// TIA Portal V15 export
// export: Created 2018-12-10T18:36:46.2365966Z, ExportSetting WithDefaults, WithReadOnly, DisplayName Totally Integrated Automation Portal, DisplayVersion V15 Update 2, DisplayName TIA Portal Openness, DisplayVersion V15 Update 2, DisplayName STEP 7 Professional, DisplayVersion V15 Update 2, DisplayName STEP 7 Safety, DisplayVersion V15, DisplayName WinCC Professional, DisplayVersion V15 Update 2, DisplayName SIMATIC Visualization Architect, DisplayVersion V15 Update 1
DATA_BLOCK "FGDB_ROBNAME@FlowDrill"   // DB118
TITLE = Tehchnology flow drill / Technologie übergreifendes Gerät
{ S7_Optimized_Access := 'FALSE' }
AUTHOR : integra
FAMILY : SUB
VERSION : 0.1
// stored: AutoNumber true, CodeModifiedDate 2018-02-20T07:56:40.7852281Z, CompileDate 2018-02-20T10:24:49.1738274Z, CreationDate 2017-02-23T12:13:10.5636609Z, DBAccessibleFromOPCUA true, InstanceOfName iSF_TECH_ROBOT_FLOW_DRILL_SCREWING, InstanceOfNumber 24, InstanceOfType FB, InterfaceModifiedDate 2018-02-19T12:53:42.2863137Z, IsConsistent true, IsKnowHowProtected false, ModifiedDate 2018-02-20T07:56:40.7852281Z, ParameterModified 2018-02-19T12:53:31.0081644Z, StructureModified 2018-02-19T12:53:42.2863137Z, UDAEnableTagReadback false
"iSF_TECH_ROBOT_FLOW_DRILL_SCREWING"
   // VAR_INPUT
   //    fct : Int;
   //    safetyStop : Bool;
   //    functionPoint : String[6];
   //    identType : String[12];
   // END_VAR
   // VAR_OUTPUT
   //    counterParts : Int;
   //    counterNIOpoints : Int;
   //    counterIOpoints : Int;
   //    fault : Bool;
   // END_VAR
   // VAR_IN_OUT
   //    IfcFGExternal : "iUDT_IFC_SYS_EXTERNAL_ALARM";
   //    IfcTECH : "iUDT_IFC_ROBOT_TECH";
   //    IfcAcyclicdata : "iUDT_IFC_ROBOT_ACYCLICDATA";
   //    ident : Variant;
   //    IfcTLG : "iUDT_IFC_TLG";
   //    TLG_MQDV : "iUDT_TLG_MQDV_ROBOT";
   //    TLG_ENEV : "iUDT_TLG_ENEV";
   //    In_PI_TECH : "iUDT_PI_ROBOT_ADRxx48_TECH";
   //    Out_PO_TECH : "iUDT_PO_ROBOT_ADRxx48_TECH";
   // END_VAR
   // VAR RETAIN
   //    F : Struct
   //       wrongID : Bool;
   //       system : Bool;
   //       processStop : Bool;
   //       fehlerSystem : Bool;
   //       plus : Bool;
   //    END_STRUCT;
   //    W : Struct
   //       errorProzess : Bool;
   //       warningLimit : Bool;
   //       quantityMax : Bool;
   //       levelControl : Bool;
   //    END_STRUCT;
   //    Masks : Struct
   //       disableFault1_8 : Byte;
   //       prodRelevantFault1_8 : Byte;
   //       prodRelevantWarningt_1_8 : Byte;
   //    END_STRUCT;
   //    LastState : Struct
   //       fault1_8 : Byte;
   //       warning_1_8 : Byte;
   //    END_STRUCT;
   //    Tmr : Struct
   //       s1 { S7_SetPoint := 'True'} : Int;
   //       a1 : Int;
   //    END_STRUCT;
   //    TmrB : Struct
   //       "1_EnableDelayTime" : Bool;
   //       "1_RunDelayTime" : Bool;
   //       "1_DoneDelayTime" : Bool;
   //    END_STRUCT;
   //    TECH : Struct
   //       ID : Byte;
   //       System_OK : Bool;
   //       qualityOK : Bool;
   //       qualityNOK : Bool;
   //       ready : Bool;
   //       automaticActive : Bool;
   //       STO : Bool;
   //       prozessStop : Bool;
   //       errorProzess : Bool;
   //       errorSystem : Bool;
   //       warningLimit : Bool;
   //       quantityMax : Bool;
   //       levelControl : Bool;
   //       operatorProtection : Bool;
   //       confirmAccess : Bool;
   //       technoBit15 : Bool;
   //       technoBit16 : Bool;
   //       technoBit17 : Bool;
   //       technoBit18 : Bool;
   //       technoBit19 : Bool;
   //       technoBit20 : Bool;
   //       technoBit21 : Bool;
   //       technoBit22 : Bool;
   //       technoBit23 : Bool;
   //       technoBit24 : Bool;
   //       technoBit25 : Bool;
   //       technoBit26 : Bool;
   //       technoBit27 : Bool;
   //       technoBit28 : Bool;
   //       technoBit29 : Bool;
   //       technoBit30 : Bool;
   //       technoBit31 : Bool;
   //       technoBit32 : Bool;
   //       technoBit33 : Bool;
   //       technoBit34 : Bool;
   //       technoBit35 : Bool;
   //       technoBit36 : Bool;
   //       technoBit37 : Bool;
   //       technoBit38 : Bool;
   //       technoBit39 : Bool;
   //       technoBit40 : Bool;
   //    END_STRUCT;
   //    PLUS : "iIF_ROBOT_PLUS";
   // END_VAR
BEGIN
END_DATA_BLOCK
